PROGRAM MAIN
VAR
    ControlSource_HMI : FB_ControlSource_HMI_Machine;
    Seedra          : FB_Machine := (Name := 'Seedra_');
    InitComplete      : BOOL;

    //Debug testing Recipe manager
    Value1 : INT;
    Value2 : INT;
END_VAR

CyclicLogic();

METHOD CyclicLogic
VAR_INPUT
END_VAR
IF NOT InitComplete THEN
    InitComplete := Initialize();
    RETURN;
END_IF

//Machine support HMI & Production Monitor
ControlSource_HMI.CyclicLogic();

//Machine Cyclic Logic
Seedra.CyclicLogic();
END_METHOD

METHOD Initialize : BOOL
VAR_INPUT
END_VAR
//Top level machine initialization should happen here, in the main initialization method. Each subsequent "layer" of modules will be named within their respective "parent" intialize method
_AppInfo.KeepOutputsOnBP := TRUE;
IF NOT ControlSource_HMI.Registered THEN
    Seedra.RegisterExternalController(ControlSource_HMI);
END_IF

ControlSource_HMI.CyclicLogic();
Initialize := TRUE;
END_METHOD

END_PROGRAM

(* stored: Version 1.1.0.1
   POU MAIN: Id {0a415e5e-1cd5-4d94-8552-fcd14dfd2571}, SpecialFunc None
   Method CyclicLogic: Id {8bb74a65-86fc-4043-b45c-8f31846cbc32}
   Method Initialize: Id {b0a02fad-0cef-4243-8118-97702c63fa8f} *)
